Staubli VAL3: getSize_num.pgx

public program getSize_num(num& x_nSize[] (dimensions=1))
begin
  // get the size for the counter
  x_nSize=size(cCount)
  // get the size for the aCounter
  x_nSize=x_nSize+size(aCount)
end
